(* CoDeSys 2.3.8.1 project: Test.pro *)
(* Libraries: ComService.lib 21.5.09 15:28:28, SysLibCom.lib 26.10.04 15:15:20, ANALYZATION.LIB 5.10.99 10:05:06, ModBus.lib 27.5.09 10:22:38, SYSLIBTIME.lib*23.9.04 11:11:36, Standard.lib 4.10.05 12:14:46, IecSfc.lib 13.4.06 16:51:28, SYSLIBCALLBACK.LIB 16.4.07 17:52:46 *)

(* POU PLC_PRG, ST *)
PROGRAM PLC_PRG
VAR
	send1_modbus:MB_WR_SNG_REG; (*функция 06 - запись параметра*)

	COM_SERVICE1: COM_SERVICE; (*ФБ открытия порта*)
	Buffer: ARRAY[0..255] OF BYTE; (* байтовый буфер данных *)
	cmpl: BOOL; (* признак завершения операции *)
	port_opened: BYTE := 0; (*состояние порта*)
	Init: BOOL; (* признак инициализации пользовательской программы *)
	Settings:COMSETTINGS; (* настройки последовательного порта *)
	com_num: PORTS:=COM1; (*0 - RS-485, 1 - RS-232*)
	enabl: BOOL; (*состояние работы блока*)
	err: INT; (*номер ошибки*)
	TimeOut: TIME:=T#50ms; (*таймаут*)
	Exception: BYTE;
	DataSize: WORD;
	master1: BYTE;
	t: DWORD; (*переменная для организации счетчика*)
	A: WORD := 0; (*счетчик*)
	f1:DINT:=65; (*Записываемый параметр типа DINT*)
	f2:REAL:=12.7; (*Записываемый параметр типа REAL*)
	ptr_f2:POINTER TO BYTE;
END_VAR
(*Организуем счетчик, что бы передавать эти данные по сети*)
t:=t+1;
IF (t MOD 1000)=0 THEN
	A := A + 1;
	IF A > 9999 THEN
		A := 0;
	END_IF
END_IF

(*Устанавливаем настройки COM-порта*)
IF port_opened=0 THEN
	Settings.Port:=com_num; (*номер COM-порта*)
	Settings.dwBaudRate:=9600; (*скорость*)
	Settings.byParity:=1;
	Settings.dwTimeout:=0;
	Settings.byStopBits:=1;
	Settings.dwBufferSize:=0;
	Settings.dwScan:=0;
END_IF
(*Открываем COM-порт*)
COM_SERVICE1(Enable:=(port_opened=0) , Settings:=Settings , Task:=OPEN_TSK );
(*Если COM-порт открыт, то переходим к приему и передачи данных *)
IF COM_SERVICE1.ready THEN
	port_opened:=2;
END_IF
IF port_opened=2 THEN (*Удачно проинициализировали*)
CASE master1 OF
0: (* функция 06 - запись параметра типа Int в прибор с адресом 1 в регистр 0*)
send1_modbus(
	Enable:=enabl , (* разрешение работы блока *)
	Mode:=MB_RTU, (*режим передачи*)
	DevAddr:=1 , (*адрес*)
	RegAddr:=0 , (*регистр*)
	Value:=A, (*значение переменной, которое надо передать*)
	ComHandle:= Settings.Port, (*номер сом-порта*)
	TimeOut:=TimeOut , (*таймаут T#50ms*)
	Complete=>cmpl , (* скопировать признак завершения операции *)
	Exception=>err ); (* скопировать регистр ошибок *)
(*если установлен признак завершения операции, то *)
IF cmpl THEN
	master1:=0; (*переходим к выполнению следующего блока*)
END_IF
END_CASE
	IF enabl = FALSE THEN
		enabl := TRUE;
	END_IF
	IF err <> 0 THEN
		enabl := FALSE;
	END_IF
END_IF
END_PROGRAM
